{attribute 'qualified_only'}
{attribute 'strict'}
{attribute 'to_string'}
TYPE E_MoveState :
(
    IDLING:=0,
    INIT:=10,
    STARTED:=20,
    IN_PROGRESS :=30,
    REACHED:=40,
    INTERRUPTED:=50,
    DONE:=60,
    ERROR:=-99
);
END_TYPE

(* stored: Version 1.1.0.1
   DUT E_MoveState: Id {b8df697a-8c28-4be4-a4a4-3221be1ce7a3} *)
